// TIA Portal V15.1 export
// export: Created 2024-06-21T08:41:15.2756502Z, ExportSetting WithDefaults, DisplayName Totally Integrated Automation Portal, DisplayVersion V15.1 Update 5, DisplayName TIA Portal Openness, DisplayVersion V15.1 Update 5, DisplayName SINAMICS Startdrive Advanced, DisplayVersion V15.1, DisplayName G130, G150, S120, S150, SINAMICS MV, S210, DisplayVersion V15.1, DisplayName G110M, G120, G120C, G120D, G120P, DisplayVersion V15.1, DisplayName STEP 7 Professional, DisplayVersion V15.1 Update 5, DisplayName STEP 7 Safety, DisplayVersion V15.1, DisplayName WinCC Professional, DisplayVersion V15.1 Update 5, DisplayName SIMATIC Visualization Architect, DisplayVersion V15.1
FUNCTION_BLOCK "LGBChain2W1S-FC302PN"   // FB6603, FBD
TITLE = LGBChain2W1S-FC302PN
{ S7_Optimized_Access := 'FALSE' }
VERSION : 0.1
// stored: AutoNumber false, IsIECCheckEnabled false, SetENOAutomatically False, UDAEnableTagReadback false
   VAR_INPUT
      I_ExitDet { ExternalAccessible := 'False'; ExternalVisible := 'False'; ExternalWritable := 'False'} : Bool;   // Stop Detection set
      I_EntranceDet { ExternalAccessible := 'False'; ExternalVisible := 'False'; ExternalWritable := 'False'} : Bool;   // Stop Detection Reset
      I_StopDetPrev { ExternalAccessible := 'False'; ExternalVisible := 'False'; ExternalWritable := 'False'} : Bool;   // Stop Detection previous conveyor
      I_ChainTensionLDet { ExternalAccessible := 'False'; ExternalVisible := 'False'; ExternalWritable := 'False'} : Bool;   // Chain Tension left detection
      I_ChainTensionRDet { ExternalAccessible := 'False'; ExternalVisible := 'False'; ExternalWritable := 'False'} : Bool;   // Chain Tension Right detection
      I_SlackChainDet { ExternalAccessible := 'False'; ExternalVisible := 'False'; ExternalWritable := 'False'} : Bool;   // Slack Chain detection
      I_TrfInSetBegin { ExternalAccessible := 'False'; ExternalVisible := 'False'; ExternalWritable := 'False'} : Bool;   // Load Begin: condition to start transfer IN set
      I_TrfInSetIntlkOk { ExternalAccessible := 'False'; ExternalVisible := 'False'; ExternalWritable := 'False'} : Bool;   // Transfer IN Interlock Set OK
      I_TrfOutSetBegin { ExternalAccessible := 'False'; ExternalVisible := 'False'; ExternalWritable := 'False'} : Bool;   // Unload Begin: condition to start transfer OUT set
      I_TrfOutSetIntlkOk { ExternalAccessible := 'False'; ExternalVisible := 'False'; ExternalWritable := 'False'} : Bool;   // Transfer Out Interlock Set OK
      I_TrfInSetRdyDlv { ExternalAccessible := 'False'; ExternalVisible := 'False'; ExternalWritable := 'False'} : Bool;   // Ready to deliver: Signal from previous object set
      I_TrfInSetTM { ExternalAccessible := 'False'; ExternalVisible := 'False'; ExternalWritable := 'False'} : Bool;   // Transfer busy signal from previous equipement set
      I_TrfOutSetRdyRcv { ExternalAccessible := 'False'; ExternalVisible := 'False'; ExternalWritable := 'False'} : Bool;   // Ready to Receive: Signal from next object set
      I_TrfOutSetArrived { ExternalAccessible := 'False'; ExternalVisible := 'False'; ExternalWritable := 'False'} : Bool;   // Body Arrived: Signal from next object Set
      I_PBSet { ExternalAccessible := 'False'; ExternalVisible := 'False'; ExternalWritable := 'False'} : Bool;   // Push button for manual movement (on local panel) set
      I_PBReset { ExternalAccessible := 'False'; ExternalVisible := 'False'; ExternalWritable := 'False'} : Bool;   // Push button for manual movement (on local panel) Reset
      I_ManInfeedAllowedSet { ExternalAccessible := 'False'; ExternalVisible := 'False'; ExternalWritable := 'False'} : Bool;   // Manual Infeed Allowed Set (without PushButton)
      I_ManInfeedAllowedRes { ExternalAccessible := 'False'; ExternalVisible := 'False'; ExternalWritable := 'False'} : Bool;   // Manual Infeed Allowed Reset (without PushButton)
      I_MotorProtection { ExternalAccessible := 'False'; ExternalVisible := 'False'; ExternalWritable := 'False'} : Bool;   // Motorprotection
      I_BrakeProtection { ExternalAccessible := 'False'; ExternalVisible := 'False'; ExternalWritable := 'False'} : Bool;   // Brake protection
      I_SafetySwitch { ExternalAccessible := 'False'; ExternalVisible := 'False'; ExternalWritable := 'False'} : Bool;   // Safety switch
      I_ReleaseBrakeMot { ExternalAccessible := 'False'; ExternalVisible := 'False'; ExternalWritable := 'False'} : Bool;   // Release brake motor
      I_SafetyOk { ExternalAccessible := 'False'; ExternalVisible := 'False'; ExternalWritable := 'False'} : Bool;   // Safety Ok
      I_MotionStopOk { ExternalAccessible := 'False'; ExternalVisible := 'False'; ExternalWritable := 'False'} : Bool;   // Safety Ok / The motion stop is Ok
      I_ProductionStop { ExternalAccessible := 'False'; ExternalVisible := 'False'; ExternalWritable := 'False'} : Bool;   // Production Stop
      I_ExtStartConveyor { ExternalAccessible := 'False'; ExternalVisible := 'False'; ExternalWritable := 'False'} : Bool;   // External Start Conveyor
      I_SpeedSetPoint { ExternalAccessible := 'False'; ExternalVisible := 'False'; ExternalWritable := 'False'} : Real;   // Speed set point value motor (cm/min)
      I_ChainEmptyTime { ExternalAccessible := 'False'; ExternalVisible := 'False'; ExternalWritable := 'False'} : DInt;   // Time to empty Chain (Msec)
   END_VAR
   VAR_OUTPUT
      O_Active { ExternalAccessible := 'False'; ExternalVisible := 'False'; ExternalWritable := 'False'} : Bool;   // Chain is Active
      O_TrfInSetRdyRcv { ExternalAccessible := 'False'; ExternalVisible := 'False'; ExternalWritable := 'False'} : Bool;   // Ready to Receive: Signal to previous object set
      O_TrfInSetArrived { ExternalAccessible := 'False'; ExternalVisible := 'False'; ExternalWritable := 'False'} : Bool;   // Body Arrived: Signal to previous object Set
      O_TrfOutSetRdyDlv { ExternalAccessible := 'False'; ExternalVisible := 'False'; ExternalWritable := 'False'} : Bool;   // Ready to Deliver: Signal to next object set
      O_TrfOutSetTM { ExternalAccessible := 'False'; ExternalVisible := 'False'; ExternalWritable := 'False'} : Bool;   // Transfer: Signal to next object set
      O_TrfInSetActive { ExternalAccessible := 'False'; ExternalVisible := 'False'; ExternalWritable := 'False'} : Bool;   // Transfer in set active
      O_TrfInSetFinished { ExternalAccessible := 'False'; ExternalVisible := 'False'; ExternalWritable := 'False'} : Bool;   // Transfer in set finished
      O_TrfOutSetActive { ExternalAccessible := 'False'; ExternalVisible := 'False'; ExternalWritable := 'False'} : Bool;   // Transfer out set active
      O_TrfOutSetFinished { ExternalAccessible := 'False'; ExternalVisible := 'False'; ExternalWritable := 'False'} : Bool;   // Transfer out set finished
      O_LedRoller { ExternalAccessible := 'False'; ExternalVisible := 'False'; ExternalWritable := 'False'} : Bool;   // Led of Chain
      O_SetMotorCmd { ExternalAccessible := 'False'; ExternalVisible := 'False'; ExternalWritable := 'False'} : Bool;   // High Speed Set Command from function after Interlock
      O_ResMotorCmd { ExternalAccessible := 'False'; ExternalVisible := 'False'; ExternalWritable := 'False'} : Bool;   // High speed Reset Command from function after Interlock
      O_AlarmABCondition { ExternalAccessible := 'False'; ExternalVisible := 'False'; ExternalWritable := 'False'} : Bool;   // Alarm AB Condition
      O_AlarmA { ExternalAccessible := 'False'; ExternalVisible := 'False'; ExternalWritable := 'False'} : Bool;   // Alarm A
      O_AlarmB { ExternalAccessible := 'False'; ExternalVisible := 'False'; ExternalWritable := 'False'} : Bool;   // Alarm B
      O_AlarmC { ExternalAccessible := 'False'; ExternalVisible := 'False'; ExternalWritable := 'False'} : Bool;   // Alarm C
      O_AlarmD { ExternalAccessible := 'False'; ExternalVisible := 'False'; ExternalWritable := 'False'} : Bool;   // Alarm D
      O_Occupied { ExternalAccessible := 'False'; ExternalVisible := 'False'; ExternalWritable := 'False'} : Bool;   // Chain Occupied
      O_ActualSpeed { ExternalAccessible := 'False'; ExternalVisible := 'False'; ExternalWritable := 'False'} : Int;   // Actual speed value motor (cm/min)
      O_ActualCurrent { ExternalAccessible := 'False'; ExternalVisible := 'False'; ExternalWritable := 'False'} : Real;   // Actual Current value motor (A)
      H_AlarmDWord { ExternalAccessible := 'False'; ExternalVisible := 'False'; ExternalWritable := 'False'} : DWord;   // HMI Animation
   END_VAR
   VAR_IN_OUT
      C_TimeCheckSpeedOK { ExternalAccessible := 'False'; ExternalVisible := 'False'; ExternalWritable := 'False'} : DInt := 2000;   // Time check speed OK
      IO_Modes : "Modes";   // Modes
      H_HMI : "H_HMI";   // Animation
      "H_GBChain2W1S-FC302PN" : "H_GBChain2W1S-FC302PN";   // Animation
      C_Config : "RollerConvConfig";   // Config
   END_VAR
   VAR DB_SPECIFIC
      H_FncSelInHMI { ExternalAccessible := 'False'; ExternalVisible := 'False'; ExternalWritable := 'False'} : Bool;
      AB_ChainTensionLAlm { ExternalAccessible := 'False'; ExternalVisible := 'False'; ExternalWritable := 'False'} : Bool;   // Alarm Chain Tension Left
      AB_ChainTensionRAlm { ExternalAccessible := 'False'; ExternalVisible := 'False'; ExternalWritable := 'False'} : Bool;   // Alarm Chain Tension Right
      AB_SlackChainAlm { ExternalAccessible := 'False'; ExternalVisible := 'False'; ExternalWritable := 'False'} : Bool;   // Alarm Slack Chain
      AC_TrfOutSetOverTime { ExternalAccessible := 'False'; ExternalVisible := 'False'; ExternalWritable := 'False'} : Bool;   // Timeout Transport Out Set
      AD_TrfOutSetInterlock { ExternalAccessible := 'False'; ExternalVisible := 'False'; ExternalWritable := 'False'} : Bool;   // Interlock Not Ok Transport Out Set
      AD_TrfInSetInterlock { ExternalAccessible := 'False'; ExternalVisible := 'False'; ExternalWritable := 'False'} : Bool;   // Interlock Not Ok Transport In Set
      AA_BusFault { ExternalAccessible := 'False'; ExternalVisible := 'False'; ExternalWritable := 'False'} : Bool;   // Drive Bus Fault
      AA_MotorProtector { ExternalAccessible := 'False'; ExternalVisible := 'False'; ExternalWritable := 'False'} : Bool;   // Motor Protection Tripped
      AA_BrakeProtection { ExternalAccessible := 'False'; ExternalVisible := 'False'; ExternalWritable := 'False'} : Bool;   // Brake Protection Tripped
      AA_SafetySwitch { ExternalAccessible := 'False'; ExternalVisible := 'False'; ExternalWritable := 'False'} : Bool;   // Safety Switch Not Ok
      AD_WarningFrqcnvMot { ExternalAccessible := 'False'; ExternalVisible := 'False'; ExternalWritable := 'False'} : Bool;   // Frequency Control FC302 Warning motor
      AB_AlarmFrqcnvMot { ExternalAccessible := 'False'; ExternalVisible := 'False'; ExternalWritable := 'False'} : Bool;   // Frequency Control FC302 Alarm motor
      AB_CurrentSensorAlm { ExternalAccessible := 'False'; ExternalVisible := 'False'; ExternalWritable := 'False'} : Bool;   // Over Current Motor
      AB_OverCurrentHHAlm { ExternalAccessible := 'False'; ExternalVisible := 'False'; ExternalWritable := 'False'} : Bool;   // Over Current Motor
      AB_OverCurrentHAlm { ExternalAccessible := 'False'; ExternalVisible := 'False'; ExternalWritable := 'False'} : Bool;   // Over Current Motor
      AB_OverCurrentLAlm { ExternalAccessible := 'False'; ExternalVisible := 'False'; ExternalWritable := 'False'} : Bool;   // Over Current Motor
      AB_OverCurrentLLAlm { ExternalAccessible := 'False'; ExternalVisible := 'False'; ExternalWritable := 'False'} : Bool;   // Over Current Motor
      AD_MotionStop { ExternalAccessible := 'False'; ExternalVisible := 'False'; ExternalWritable := 'False'} : Bool;   // Motion Stop
      AC_ConfigCalibrationAlm { ExternalAccessible := 'False'; ExternalVisible := 'False'; ExternalWritable := 'False'} : Bool;   // The Config values for Alarm Transfer time must be ALL zero or ALL different from zero
      AD_CalibrationSetWarn { ExternalAccessible := 'False'; ExternalVisible := 'False'; ExternalWritable := 'False'} : Bool;   // No High speed selected so Calibration is not possible for SET direction
      SafetyOk { ExternalAccessible := 'False'; ExternalVisible := 'False'; ExternalWritable := 'False'} : Bool;   // Safety Ok
      OverCurrentHAlmCond { ExternalAccessible := 'False'; ExternalVisible := 'False'; ExternalWritable := 'False'} : Bool;   // Over Current Motor
      ChainTensionLAlmCond { ExternalAccessible := 'False'; ExternalVisible := 'False'; ExternalWritable := 'False'} : Bool;   // Alarm Chain Tension Left
      ChainTensionRAlmCond { ExternalAccessible := 'False'; ExternalVisible := 'False'; ExternalWritable := 'False'} : Bool;   // Alarm Chain Tension Right
      SlackChainAlmCond { ExternalAccessible := 'False'; ExternalVisible := 'False'; ExternalWritable := 'False'} : Bool;   // Alarm Slack Chain
      MotorLoopActive { ExternalAccessible := 'False'; ExternalVisible := 'False'; ExternalWritable := 'False'} : Bool;   // Motor Loop Active
      TrfInfeedHoldSet { ExternalAccessible := 'False'; ExternalVisible := 'False'; ExternalWritable := 'False'} : Bool;   // Transfer infeed hold set direction
      TrfOutSetCmd { ExternalAccessible := 'False'; ExternalVisible := 'False'; ExternalWritable := 'False'} : Bool;   // Command after Interlock to Motor set
      TrfOutfeedHoldSet { ExternalAccessible := 'False'; ExternalVisible := 'False'; ExternalWritable := 'False'} : Bool;   // Transfer outfeed hold set direction
      TrfInSetCmd { ExternalAccessible := 'False'; ExternalVisible := 'False'; ExternalWritable := 'False'} : Bool;   // Command after Interlock to Motor set
      MotorCmdSet { ExternalAccessible := 'False'; ExternalVisible := 'False'; ExternalWritable := 'False'} : Bool;   // Command to Motorloop High Speed Set
      MotorCmdRes { ExternalAccessible := 'False'; ExternalVisible := 'False'; ExternalWritable := 'False'} : Bool;   // Command to Motorloop High Speed Reset
      TrfInSetActive { ExternalAccessible := 'False'; ExternalVisible := 'False'; ExternalWritable := 'False'} : Bool;   // Load: Active (set)
      TrfOutSetActive { ExternalAccessible := 'False'; ExternalVisible := 'False'; ExternalWritable := 'False'} : Bool;   // Unload: active (set)
      TrfOutSetFinished { ExternalAccessible := 'False'; ExternalVisible := 'False'; ExternalWritable := 'False'} : Bool;   // Unload: finished (set)
      AlarmA { ExternalAccessible := 'False'; ExternalVisible := 'False'; ExternalWritable := 'False'} : Bool;   // Alarm A
      AlarmB { ExternalAccessible := 'False'; ExternalVisible := 'False'; ExternalWritable := 'False'} : Bool;   // Alarm B
      AlarmC { ExternalAccessible := 'False'; ExternalVisible := 'False'; ExternalWritable := 'False'} : Bool;   // Alarm C
      AlarmD { ExternalAccessible := 'False'; ExternalVisible := 'False'; ExternalWritable := 'False'} : Bool;   // Alarm D
      ManLowSpdSel { ExternalAccessible := 'False'; ExternalVisible := 'False'; ExternalWritable := 'False'} : Bool;   // Low speed Selected in manual
      TrfOutSetRdyDlv { ExternalAccessible := 'False'; ExternalVisible := 'False'; ExternalWritable := 'False'} : Bool;   // Ready to Deliver: Signal to next object set
      TrfOutSetTM { ExternalAccessible := 'False'; ExternalVisible := 'False'; ExternalWritable := 'False'} : Bool;   // Transfer : Signal transfer memory to next object set
      TrfInSetTrfOutSetTM { ExternalAccessible := 'False'; ExternalVisible := 'False'; ExternalWritable := 'False'} : Bool;   // Transfer memory set
      TrfInSetRdyRcv { ExternalAccessible := 'False'; ExternalVisible := 'False'; ExternalWritable := 'False'} : Bool;   // Ready to Receive: Signal to previous object set
      TrfInSetArrived { ExternalAccessible := 'False'; ExternalVisible := 'False'; ExternalWritable := 'False'} : Bool;   // Body Arrived: Signal to previous object Set
      TrfInSetFinished { ExternalAccessible := 'False'; ExternalVisible := 'False'; ExternalWritable := 'False'} : Bool;   // Body Arrived: Signal to TrfOut module set (Reset TrfOutCmd)
      StopTrfOutSetCmd { ExternalAccessible := 'False'; ExternalVisible := 'False'; ExternalWritable := 'False'} : Bool;   // Body Arrived: Signal to previous object Set
      MotorLoopAlmCond { ExternalAccessible := 'False'; ExternalVisible := 'False'; ExternalWritable := 'False'} : Bool;   // Motor loop Alarm condition
      TrfOutSetAlmCond { ExternalAccessible := 'False'; ExternalVisible := 'False'; ExternalWritable := 'False'} : Bool;   // TrfOut set Alarm condition
      FrqReadyForOperationMot { ExternalAccessible := 'False'; ExternalVisible := 'False'; ExternalWritable := 'False'} : Bool;   // Fb motor is ready to operate motor
      ReleaseBrakeMot { ExternalAccessible := 'False'; ExternalVisible := 'False'; ExternalWritable := 'False'} : Bool;   // Req to release brake motor
      ChainStop { ExternalAccessible := 'False'; ExternalVisible := 'False'; ExternalWritable := 'False'} : Bool;   // Chain stop Productions Stop
      DlvSaturation { ExternalAccessible := 'False'; ExternalVisible := 'False'; ExternalWritable := 'False'} : Bool;   // Saturation for the diliver tranfer
      AlarmABCondition { ExternalAccessible := 'False'; ExternalVisible := 'False'; ExternalWritable := 'False'} : Bool;   // Alarm AB Condition
      HighSpeedMot { ExternalAccessible := 'False'; ExternalVisible := 'False'; ExternalWritable := 'False'} : Real;   // High speed Value (set-up %) Motor
      ActualSpeed { ExternalAccessible := 'False'; ExternalVisible := 'False'; ExternalWritable := 'False'} : Real;   // Actual Speed in % from FC302
      ChainEmpty { ExternalAccessible := 'False'; ExternalVisible := 'False'; ExternalWritable := 'False'} : Bool;   // Chain is Empty
      OverCurrAlarm { ExternalAccessible := 'False'; ExternalVisible := 'False'; ExternalWritable := 'False'} : Bool;
      AnInput { ExternalAccessible := 'False'; ExternalVisible := 'False'; ExternalWritable := 'False'} : Real;   // Actual Current
   END_VAR
   VAR
      _ChainEmptyTimer { ExternalAccessible := 'False'; ExternalVisible := 'False'; ExternalWritable := 'False'} : "LTimer";   // Timer
      _LTrfInSet { ExternalAccessible := 'False'; ExternalVisible := 'False'; ExternalWritable := 'False'} : "LGBTrfIn";   // FB
      _LTrfOutSet { ExternalAccessible := 'False'; ExternalVisible := 'False'; ExternalWritable := 'False'} : "LGBTrfOut";   // FB
      _Motor { ExternalAccessible := 'False'; ExternalVisible := 'False'; ExternalWritable := 'False'} : "LGBMotor2W2S-FC302PN";
      _MotorCurrent : "LAnInput6Lim";
      _ChainTensionLeft { ExternalAccessible := 'False'; ExternalVisible := 'False'; ExternalWritable := 'False'} : "L1AlarmMultiIn";
      _ChainTensionRight { ExternalAccessible := 'False'; ExternalVisible := 'False'; ExternalWritable := 'False'} : "L1AlarmMultiIn";
      _ChainSlack { ExternalAccessible := 'False'; ExternalVisible := 'False'; ExternalWritable := 'False'} : "L1AlarmMultiIn";
   END_VAR
   VAR DB_SPECIFIC
      Reset_TP { ExternalAccessible := 'False'; ExternalVisible := 'False'; ExternalWritable := 'False'} : TP_TIME;
   END_VAR
   VAR_TEMP
      H_HMITrfInSet : "H_HMI";   // Temp
      H_HMITrfOutSet : "H_HMI";   // Temp
      H_HMIMotor : "H_HMI";   // Temp
   END_VAR
   VAR_TEMP   // added for the SCL form of the ladder/FBD networks
      _w1 : Bool;
   END_VAR
BEGIN

REGION Network 1: **** 1 - Inputs **** Safety Ok
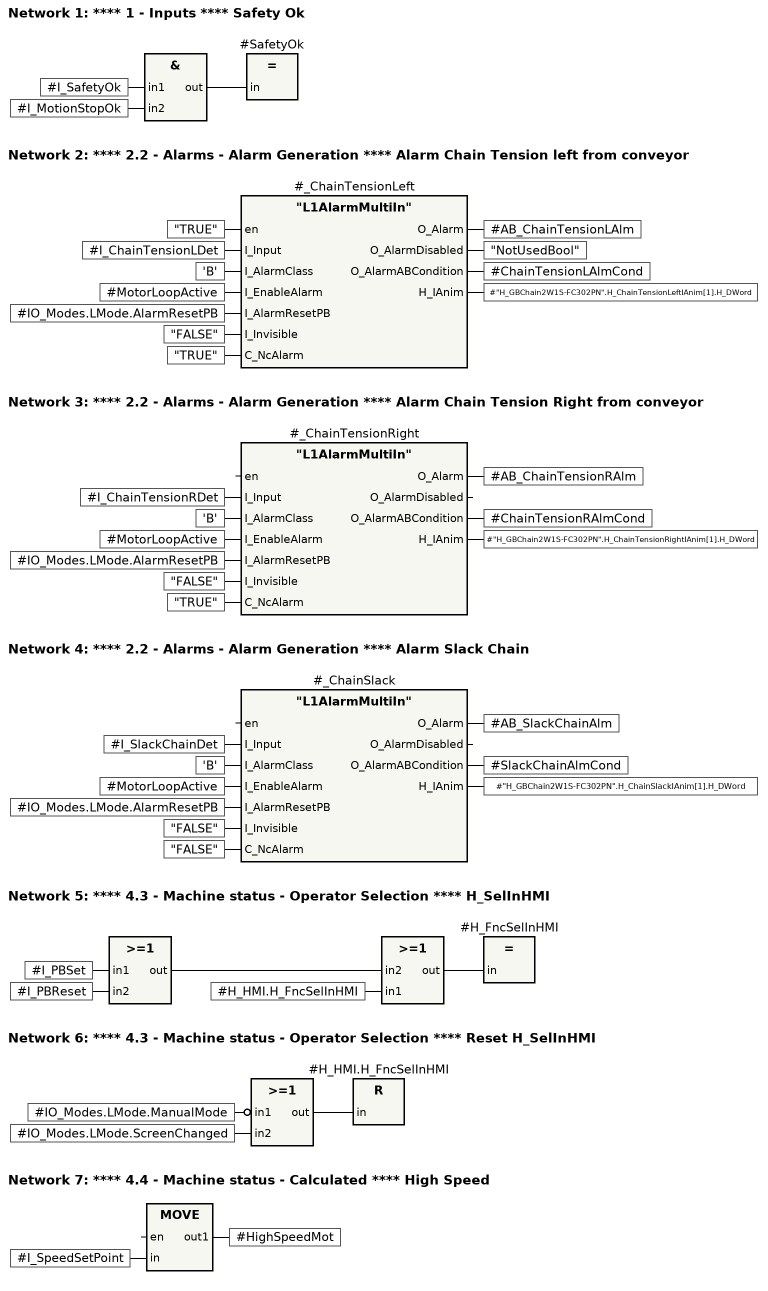
   #SafetyOk := #I_SafetyOk AND #I_MotionStopOk;
END_REGION

REGION Network 2: **** 2.2 - Alarms - Alarm Generation **** Alarm Chain Tension left from conveyor
   // Alarm Chain tension conveyor
   IF "TRUE" THEN
       #_ChainTensionLeft(I_Input := #I_ChainTensionLDet,   // "L1AlarmMultiIn"
                          I_AlarmClass := 'B',
                          I_EnableAlarm := #MotorLoopActive,
                          I_AlarmResetPB := #IO_Modes.LMode.AlarmResetPB,
                          I_Invisible := "FALSE",
                          C_NcAlarm := "TRUE",
                          O_Alarm => #AB_ChainTensionLAlm,
                          O_AlarmDisabled => "NotUsedBool",
                          O_AlarmABCondition => #ChainTensionLAlmCond,
                          H_IAnim => #"H_GBChain2W1S-FC302PN".H_ChainTensionLeftIAnim[1].H_DWord);
   END_IF;
END_REGION

REGION Network 3: **** 2.2 - Alarms - Alarm Generation **** Alarm Chain Tension Right from conveyor
   // Alarm Chain tension conveyor
   #_ChainTensionRight(I_Input := #I_ChainTensionRDet,   // "L1AlarmMultiIn"
                       I_AlarmClass := 'B',
                       I_EnableAlarm := #MotorLoopActive,
                       I_AlarmResetPB := #IO_Modes.LMode.AlarmResetPB,
                       I_Invisible := "FALSE",
                       C_NcAlarm := "TRUE",
                       O_Alarm => #AB_ChainTensionRAlm,
                       O_AlarmABCondition => #ChainTensionRAlmCond,
                       H_IAnim => #"H_GBChain2W1S-FC302PN".H_ChainTensionRightIAnim[1].H_DWord);
END_REGION

REGION Network 4: **** 2.2 - Alarms - Alarm Generation **** Alarm Slack Chain
   // Alarm Slack Chain
   #_ChainSlack(I_Input := #I_SlackChainDet,   // "L1AlarmMultiIn"
                I_AlarmClass := 'B',
                I_EnableAlarm := #MotorLoopActive,
                I_AlarmResetPB := #IO_Modes.LMode.AlarmResetPB,
                I_Invisible := "FALSE",
                C_NcAlarm := "FALSE",
                O_Alarm => #AB_SlackChainAlm,
                O_AlarmABCondition => #SlackChainAlmCond,
                H_IAnim => #"H_GBChain2W1S-FC302PN".H_ChainSlackIAnim[1].H_DWord);
END_REGION

REGION Network 5: **** 4.3 - Machine status - Operator Selection **** H_SelInHMI
   #H_FncSelInHMI := #I_PBSet OR #I_PBReset OR #H_HMI.H_FncSelInHMI;
END_REGION

REGION Network 6: **** 4.3 - Machine status - Operator Selection **** Reset H_SelInHMI
   // Reset H_SelInHMI
   IF NOT #IO_Modes.LMode.ManualMode OR #IO_Modes.LMode.ScreenChanged THEN
       #H_HMI.H_FncSelInHMI := FALSE;
   END_IF;
END_REGION

REGION Network 7: **** 4.4 - Machine status - Calculated **** High Speed
   #HighSpeedMot := #I_SpeedSetPoint;
END_REGION

REGION Network 8: **** 4.4 - Machine status - Calculated **** High Speed Motor to high
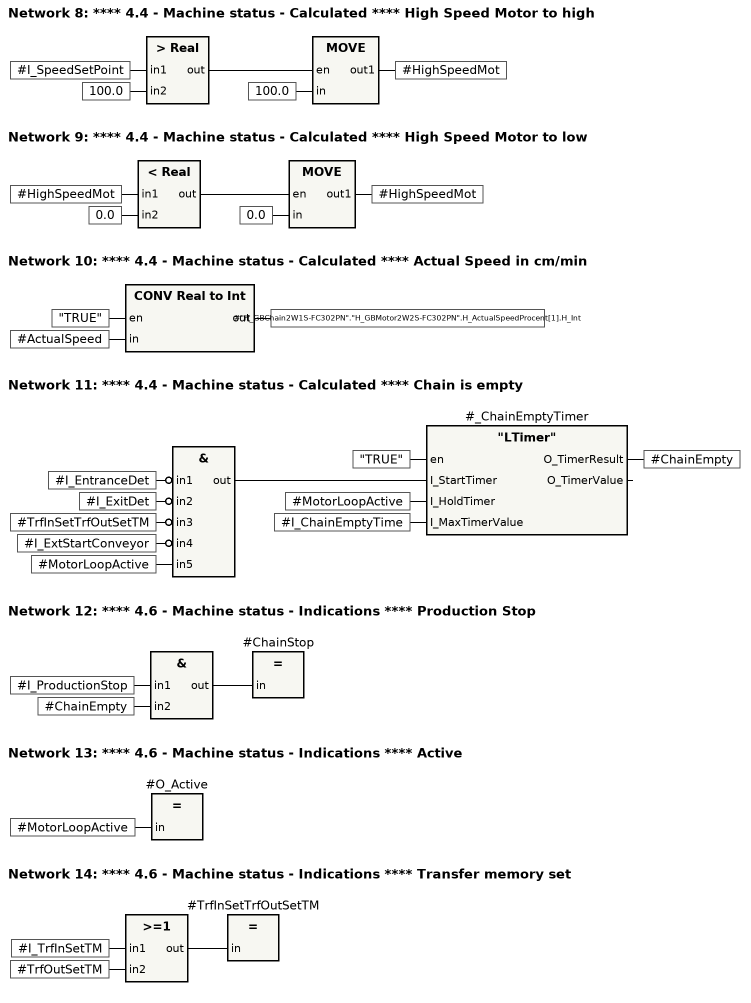
   IF #I_SpeedSetPoint > 100.0 THEN #HighSpeedMot := 100.0; END_IF;
END_REGION

REGION Network 9: **** 4.4 - Machine status - Calculated **** High Speed Motor to low
   IF #HighSpeedMot < 0.0 THEN #HighSpeedMot := 0.0; END_IF;
END_REGION

REGION Network 10: **** 4.4 - Machine status - Calculated **** Actual Speed in cm/min
   // Actual Speed in cm/min
   IF "TRUE" THEN
       #"H_GBChain2W1S-FC302PN"."H_GBMotor2W2S-FC302PN".H_ActualSpeedProcent[1].H_Int := REAL_TO_INT(#ActualSpeed);
   END_IF;
END_REGION

REGION Network 11: **** 4.4 - Machine status - Calculated **** Chain is empty
   // Chain is empty when chain is running and no detection is activated during the preset time
   IF "TRUE" THEN
       #_ChainEmptyTimer(I_StartTimer := NOT #I_EntranceDet AND NOT #I_ExitDet AND NOT #TrfInSetTrfOutSetTM AND NOT #I_ExtStartConveyor AND #MotorLoopActive,   // "LTimer"
                         I_HoldTimer := #MotorLoopActive,
                         I_MaxTimerValue := #I_ChainEmptyTime,
                         O_TimerResult => #ChainEmpty);
   END_IF;
END_REGION

REGION Network 12: **** 4.6 - Machine status - Indications **** Production Stop
   #ChainStop := #I_ProductionStop AND #ChainEmpty;
END_REGION

REGION Network 13: **** 4.6 - Machine status - Indications **** Active
   // Active
   #O_Active := #MotorLoopActive;
END_REGION

REGION Network 14: **** 4.6 - Machine status - Indications **** Transfer memory set
   // Transfer memory set
   #TrfInSetTrfOutSetTM := #I_TrfInSetTM OR #TrfOutSetTM;
END_REGION

REGION Network 15: **** 4.6 - Machine Status - Indication **** Entrance Det
   // Entrance Det
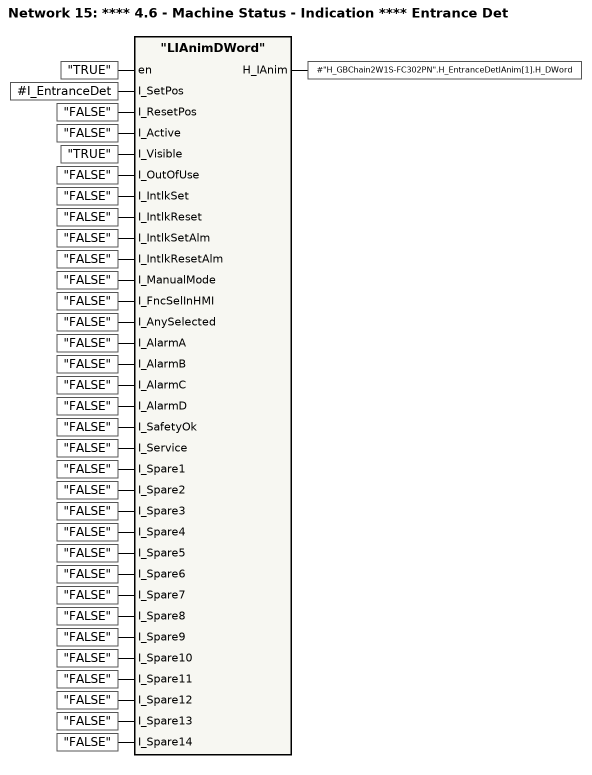
   IF "TRUE" THEN
       "LIAnimDWord"(I_SetPos := #I_EntranceDet,
                     I_ResetPos := "FALSE",
                     I_Active := "FALSE",
                     I_Visible := "TRUE",
                     I_OutOfUse := "FALSE",
                     I_IntlkSet := "FALSE",
                     I_IntlkReset := "FALSE",
                     I_IntlkSetAlm := "FALSE",
                     I_IntlkResetAlm := "FALSE",
                     I_ManualMode := "FALSE",
                     I_FncSelInHMI := "FALSE",
                     I_AnySelected := "FALSE",
                     I_AlarmA := "FALSE",
                     I_AlarmB := "FALSE",
                     I_AlarmC := "FALSE",
                     I_AlarmD := "FALSE",
                     I_SafetyOk := "FALSE",
                     I_Service := "FALSE",
                     I_Spare1 := "FALSE",
                     I_Spare2 := "FALSE",
                     I_Spare3 := "FALSE",
                     I_Spare4 := "FALSE",
                     I_Spare5 := "FALSE",
                     I_Spare6 := "FALSE",
                     I_Spare7 := "FALSE",
                     I_Spare8 := "FALSE",
                     I_Spare9 := "FALSE",
                     I_Spare10 := "FALSE",
                     I_Spare11 := "FALSE",
                     I_Spare12 := "FALSE",
                     I_Spare13 := "FALSE",
                     I_Spare14 := "FALSE",
                     H_IAnim => #"H_GBChain2W1S-FC302PN".H_EntranceDetIAnim[1].H_DWord);
   END_IF;
END_REGION

REGION Network 16: **** 4.6 - Machine Status - Indication **** Exit Det
   // Exit Det
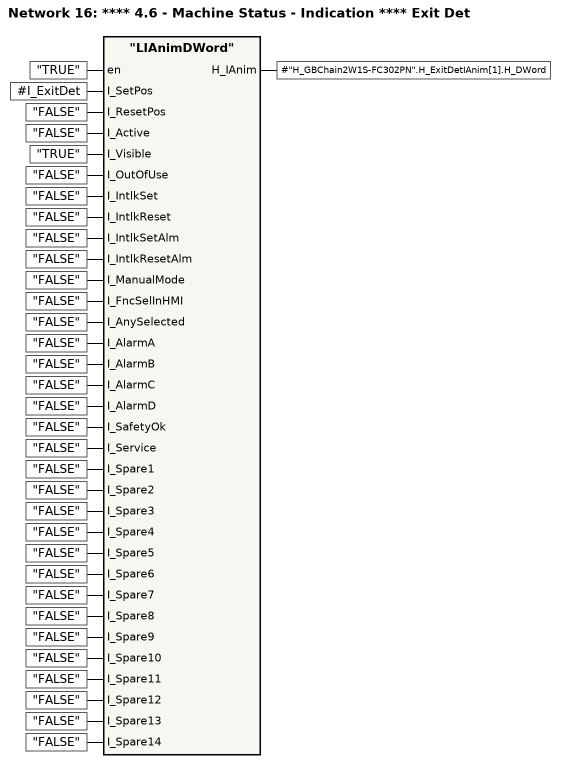
   IF "TRUE" THEN
       "LIAnimDWord"(I_SetPos := #I_ExitDet,
                     I_ResetPos := "FALSE",
                     I_Active := "FALSE",
                     I_Visible := "TRUE",
                     I_OutOfUse := "FALSE",
                     I_IntlkSet := "FALSE",
                     I_IntlkReset := "FALSE",
                     I_IntlkSetAlm := "FALSE",
                     I_IntlkResetAlm := "FALSE",
                     I_ManualMode := "FALSE",
                     I_FncSelInHMI := "FALSE",
                     I_AnySelected := "FALSE",
                     I_AlarmA := "FALSE",
                     I_AlarmB := "FALSE",
                     I_AlarmC := "FALSE",
                     I_AlarmD := "FALSE",
                     I_SafetyOk := "FALSE",
                     I_Service := "FALSE",
                     I_Spare1 := "FALSE",
                     I_Spare2 := "FALSE",
                     I_Spare3 := "FALSE",
                     I_Spare4 := "FALSE",
                     I_Spare5 := "FALSE",
                     I_Spare6 := "FALSE",
                     I_Spare7 := "FALSE",
                     I_Spare8 := "FALSE",
                     I_Spare9 := "FALSE",
                     I_Spare10 := "FALSE",
                     I_Spare11 := "FALSE",
                     I_Spare12 := "FALSE",
                     I_Spare13 := "FALSE",
                     I_Spare14 := "FALSE",
                     H_IAnim => #"H_GBChain2W1S-FC302PN".H_ExitDetIAnim[1].H_DWord);
   END_IF;
END_REGION

REGION Network 17: **** 4.6 - Machine Status - Indication **** Icon Animation
   // Icon Animation
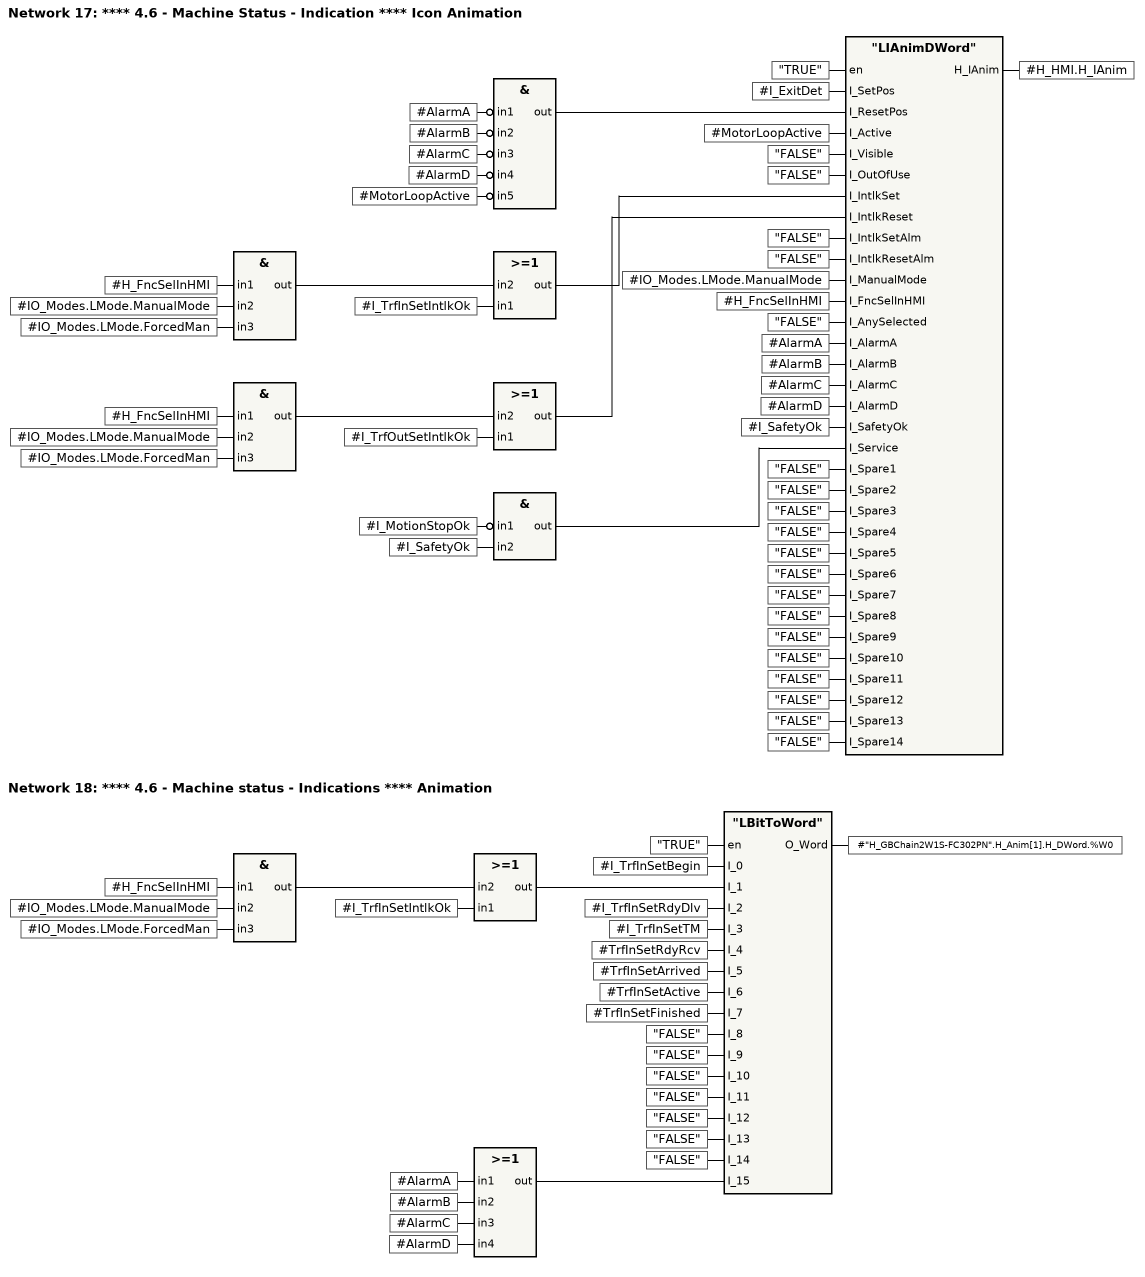
   IF "TRUE" THEN
       "LIAnimDWord"(I_SetPos := #I_ExitDet,
                     I_ResetPos := NOT #AlarmA AND NOT #AlarmB AND NOT #AlarmC AND NOT #AlarmD AND NOT #MotorLoopActive,
                     I_Active := #MotorLoopActive,
                     I_Visible := "FALSE",
                     I_OutOfUse := "FALSE",
                     I_IntlkSet := (#H_FncSelInHMI AND #IO_Modes.LMode.ManualMode AND #IO_Modes.LMode.ForcedMan) OR #I_TrfInSetIntlkOk,
                     I_IntlkReset := (#H_FncSelInHMI AND #IO_Modes.LMode.ManualMode AND #IO_Modes.LMode.ForcedMan) OR #I_TrfOutSetIntlkOk,
                     I_IntlkSetAlm := "FALSE",
                     I_IntlkResetAlm := "FALSE",
                     I_ManualMode := #IO_Modes.LMode.ManualMode,
                     I_FncSelInHMI := #H_FncSelInHMI,
                     I_AnySelected := "FALSE",
                     I_AlarmA := #AlarmA,
                     I_AlarmB := #AlarmB,
                     I_AlarmC := #AlarmC,
                     I_AlarmD := #AlarmD,
                     I_SafetyOk := #I_SafetyOk,
                     I_Service := NOT #I_MotionStopOk AND #I_SafetyOk,
                     I_Spare1 := "FALSE",
                     I_Spare2 := "FALSE",
                     I_Spare3 := "FALSE",
                     I_Spare4 := "FALSE",
                     I_Spare5 := "FALSE",
                     I_Spare6 := "FALSE",
                     I_Spare7 := "FALSE",
                     I_Spare8 := "FALSE",
                     I_Spare9 := "FALSE",
                     I_Spare10 := "FALSE",
                     I_Spare11 := "FALSE",
                     I_Spare12 := "FALSE",
                     I_Spare13 := "FALSE",
                     I_Spare14 := "FALSE",
                     H_IAnim => #H_HMI.H_IAnim);
   END_IF;
END_REGION

REGION Network 18: **** 4.6 - Machine status - Indications **** Animation
   // Animation
   IF "TRUE" THEN
       "LBitToWord"(I_0 := #I_TrfInSetBegin,
                    I_1 := (#H_FncSelInHMI AND #IO_Modes.LMode.ManualMode AND #IO_Modes.LMode.ForcedMan) OR #I_TrfInSetIntlkOk,
                    I_2 := #I_TrfInSetRdyDlv,
                    I_3 := #I_TrfInSetTM,
                    I_4 := #TrfInSetRdyRcv,
                    I_5 := #TrfInSetArrived,
                    I_6 := #TrfInSetActive,
                    I_7 := #TrfInSetFinished,
                    I_8 := "FALSE",
                    I_9 := "FALSE",
                    I_10 := "FALSE",
                    I_11 := "FALSE",
                    I_12 := "FALSE",
                    I_13 := "FALSE",
                    I_14 := "FALSE",
                    I_15 := #AlarmA OR #AlarmB OR #AlarmC OR #AlarmD,
                    O_Word => #"H_GBChain2W1S-FC302PN".H_Anim[1].H_DWord.%W0);
   END_IF;
END_REGION

REGION Network 19: **** 4.6 - Machine status - Indications **** Animation
   // Animation
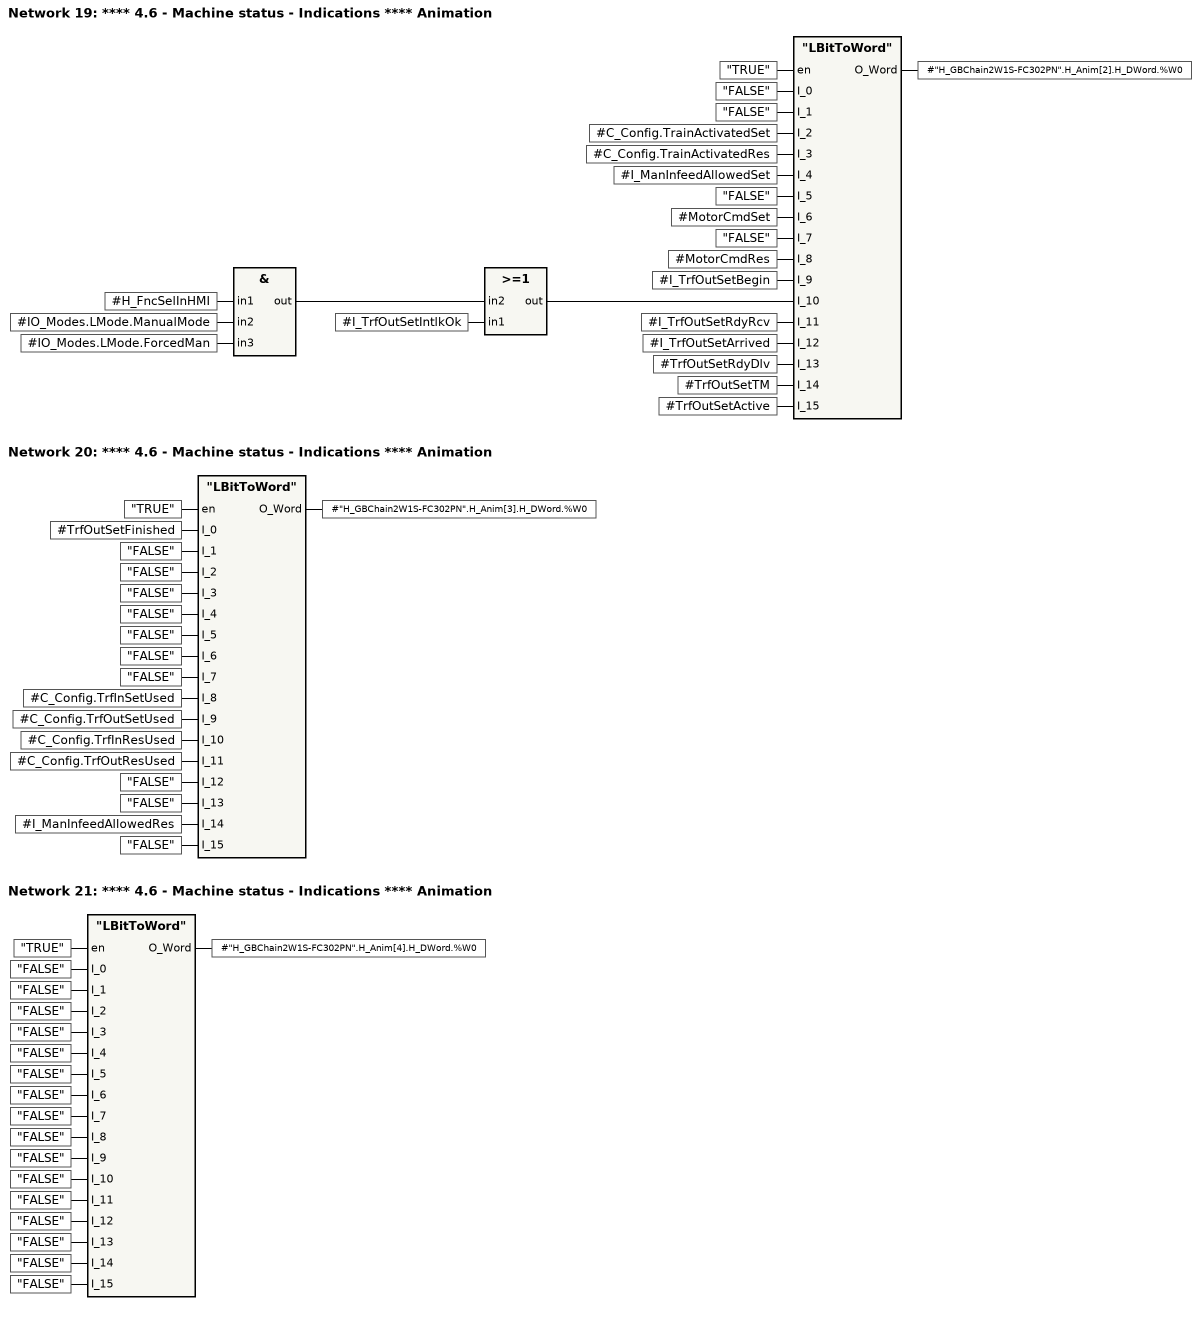
   IF "TRUE" THEN
       "LBitToWord"(I_0 := "FALSE",
                    I_1 := "FALSE",
                    I_2 := #C_Config.TrainActivatedSet,
                    I_3 := #C_Config.TrainActivatedRes,
                    I_4 := #I_ManInfeedAllowedSet,
                    I_5 := "FALSE",
                    I_6 := #MotorCmdSet,
                    I_7 := "FALSE",
                    I_8 := #MotorCmdRes,
                    I_9 := #I_TrfOutSetBegin,
                    I_10 := (#H_FncSelInHMI AND #IO_Modes.LMode.ManualMode AND #IO_Modes.LMode.ForcedMan) OR #I_TrfOutSetIntlkOk,
                    I_11 := #I_TrfOutSetRdyRcv,
                    I_12 := #I_TrfOutSetArrived,
                    I_13 := #TrfOutSetRdyDlv,
                    I_14 := #TrfOutSetTM,
                    I_15 := #TrfOutSetActive,
                    O_Word => #"H_GBChain2W1S-FC302PN".H_Anim[2].H_DWord.%W0);
   END_IF;
END_REGION

REGION Network 20: **** 4.6 - Machine status - Indications **** Animation
   // Animation
   IF "TRUE" THEN
       "LBitToWord"(I_0 := #TrfOutSetFinished,
                    I_1 := "FALSE",
                    I_2 := "FALSE",
                    I_3 := "FALSE",
                    I_4 := "FALSE",
                    I_5 := "FALSE",
                    I_6 := "FALSE",
                    I_7 := "FALSE",
                    I_8 := #C_Config.TrfInSetUsed,
                    I_9 := #C_Config.TrfOutSetUsed,
                    I_10 := #C_Config.TrfInResUsed,
                    I_11 := #C_Config.TrfOutResUsed,
                    I_12 := "FALSE",
                    I_13 := "FALSE",
                    I_14 := #I_ManInfeedAllowedRes,
                    I_15 := "FALSE",
                    O_Word => #"H_GBChain2W1S-FC302PN".H_Anim[3].H_DWord.%W0);
   END_IF;
END_REGION

REGION Network 21: **** 4.6 - Machine status - Indications **** Animation
   // Animation
   IF "TRUE" THEN
       "LBitToWord"(I_0 := "FALSE",
                    I_1 := "FALSE",
                    I_2 := "FALSE",
                    I_3 := "FALSE",
                    I_4 := "FALSE",
                    I_5 := "FALSE",
                    I_6 := "FALSE",
                    I_7 := "FALSE",
                    I_8 := "FALSE",
                    I_9 := "FALSE",
                    I_10 := "FALSE",
                    I_11 := "FALSE",
                    I_12 := "FALSE",
                    I_13 := "FALSE",
                    I_14 := "FALSE",
                    I_15 := "FALSE",
                    O_Word => #"H_GBChain2W1S-FC302PN".H_Anim[4].H_DWord.%W0);
   END_IF;
END_REGION

REGION Network 22: **** 7.1 - Submodule - Non-Machine **** Analoge Input Motor Current
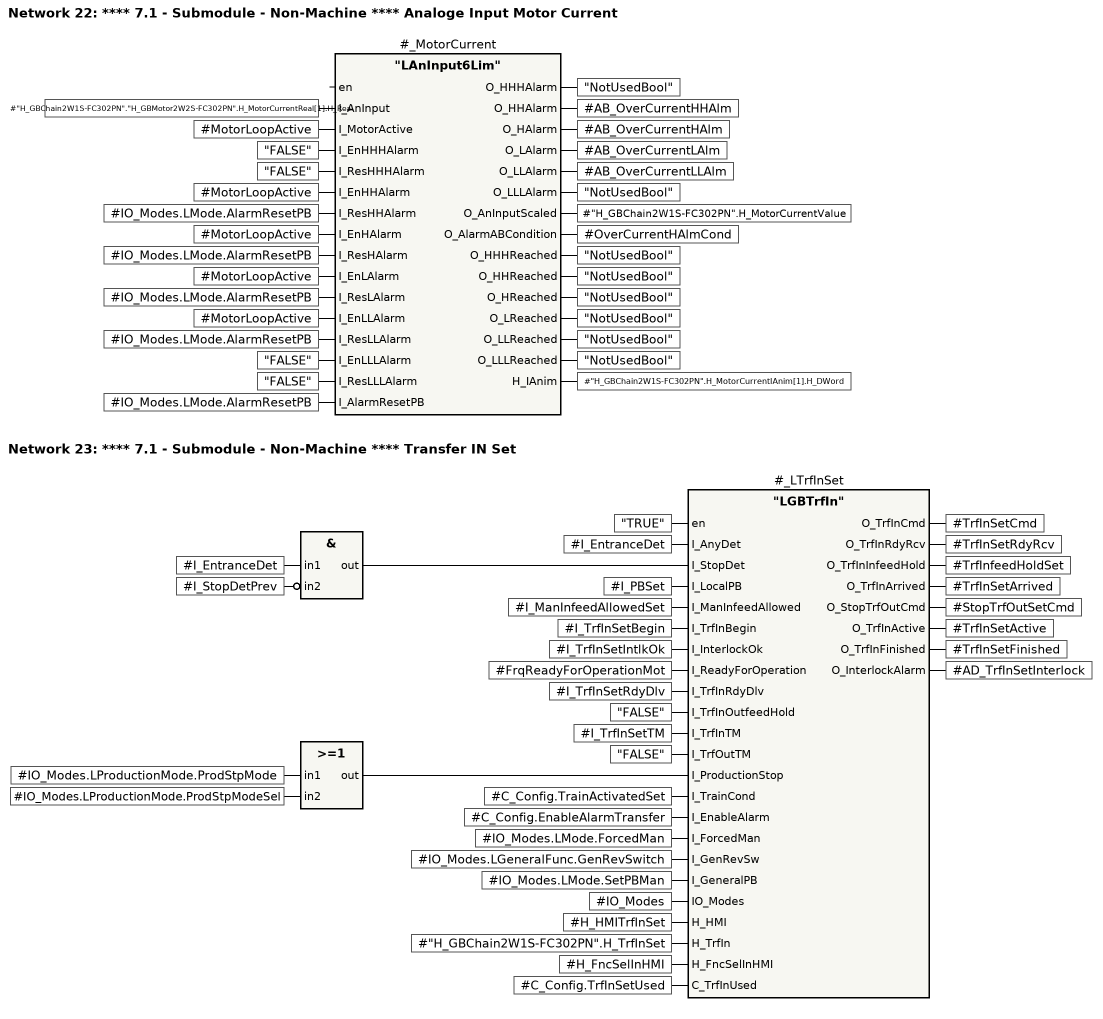
   #_MotorCurrent(I_AnInput := #"H_GBChain2W1S-FC302PN"."H_GBMotor2W2S-FC302PN".H_MotorCurrentReal[1].H_Real,   // "LAnInput6Lim"
                  I_MotorActive := #MotorLoopActive,
                  I_EnHHHAlarm := "FALSE",
                  I_ResHHHAlarm := "FALSE",
                  I_EnHHAlarm := #MotorLoopActive,
                  I_ResHHAlarm := #IO_Modes.LMode.AlarmResetPB,
                  I_EnHAlarm := #MotorLoopActive,
                  I_ResHAlarm := #IO_Modes.LMode.AlarmResetPB,
                  I_EnLAlarm := #MotorLoopActive,
                  I_ResLAlarm := #IO_Modes.LMode.AlarmResetPB,
                  I_EnLLAlarm := #MotorLoopActive,
                  I_ResLLAlarm := #IO_Modes.LMode.AlarmResetPB,
                  I_EnLLLAlarm := "FALSE",
                  I_ResLLLAlarm := "FALSE",
                  I_AlarmResetPB := #IO_Modes.LMode.AlarmResetPB,
                  O_HHHAlarm => "NotUsedBool",
                  O_HHAlarm => #AB_OverCurrentHHAlm,
                  O_HAlarm => #AB_OverCurrentHAlm,
                  O_LAlarm => #AB_OverCurrentLAlm,
                  O_LLAlarm => #AB_OverCurrentLLAlm,
                  O_LLLAlarm => "NotUsedBool",
                  O_AnInputScaled => #"H_GBChain2W1S-FC302PN".H_MotorCurrentValue,
                  O_AlarmABCondition => #OverCurrentHAlmCond,
                  O_HHHReached => "NotUsedBool",
                  O_HHReached => "NotUsedBool",
                  O_HReached => "NotUsedBool",
                  O_LReached => "NotUsedBool",
                  O_LLReached => "NotUsedBool",
                  O_LLLReached => "NotUsedBool",
                  H_IAnim => #"H_GBChain2W1S-FC302PN".H_MotorCurrentIAnim[1].H_DWord);
END_REGION

REGION Network 23: **** 7.1 - Submodule - Non-Machine **** Transfer IN Set
   // Transfer IN Set
   IF "TRUE" THEN
       #_LTrfInSet(I_AnyDet := #I_EntranceDet,   // "LGBTrfIn"
                   I_StopDet := #I_EntranceDet AND NOT #I_StopDetPrev,
                   I_LocalPB := #I_PBSet,
                   I_ManInfeedAllowed := #I_ManInfeedAllowedSet,
                   I_TrfInBegin := #I_TrfInSetBegin,
                   I_InterlockOk := #I_TrfInSetIntlkOk,
                   I_ReadyForOperation := #FrqReadyForOperationMot,
                   I_TrfInRdyDlv := #I_TrfInSetRdyDlv,
                   I_TrfInOutfeedHold := "FALSE",
                   I_TrfInTM := #I_TrfInSetTM,
                   I_TrfOutTM := "FALSE",
                   I_ProductionStop := #IO_Modes.LProductionMode.ProdStpMode OR #IO_Modes.LProductionMode.ProdStpModeSel,
                   I_TrainCond := #C_Config.TrainActivatedSet,
                   I_EnableAlarm := #C_Config.EnableAlarmTransfer,
                   I_ForcedMan := #IO_Modes.LMode.ForcedMan,
                   I_GenRevSw := #IO_Modes.LGeneralFunc.GenRevSwitch,
                   I_GeneralPB := #IO_Modes.LMode.SetPBMan,
                   IO_Modes := #IO_Modes,
                   H_HMI := #H_HMITrfInSet,
                   H_TrfIn := #"H_GBChain2W1S-FC302PN".H_TrfInSet,
                   H_FncSelInHMI := #H_FncSelInHMI,
                   C_TrfInUsed := #C_Config.TrfInSetUsed,
                   O_TrfInCmd => #TrfInSetCmd,
                   O_TrfInRdyRcv => #TrfInSetRdyRcv,
                   O_TrfInInfeedHold => #TrfInfeedHoldSet,
                   O_TrfInArrived => #TrfInSetArrived,
                   O_StopTrfOutCmd => #StopTrfOutSetCmd,
                   O_TrfInActive => #TrfInSetActive,
                   O_TrfInFinished => #TrfInSetFinished,
                   O_InterlockAlarm => #AD_TrfInSetInterlock);
   END_IF;
END_REGION

REGION Network 24: **** 7.1 - Submodule - Non-Machine **** Transfer Out Set
   // Transfer Out Set
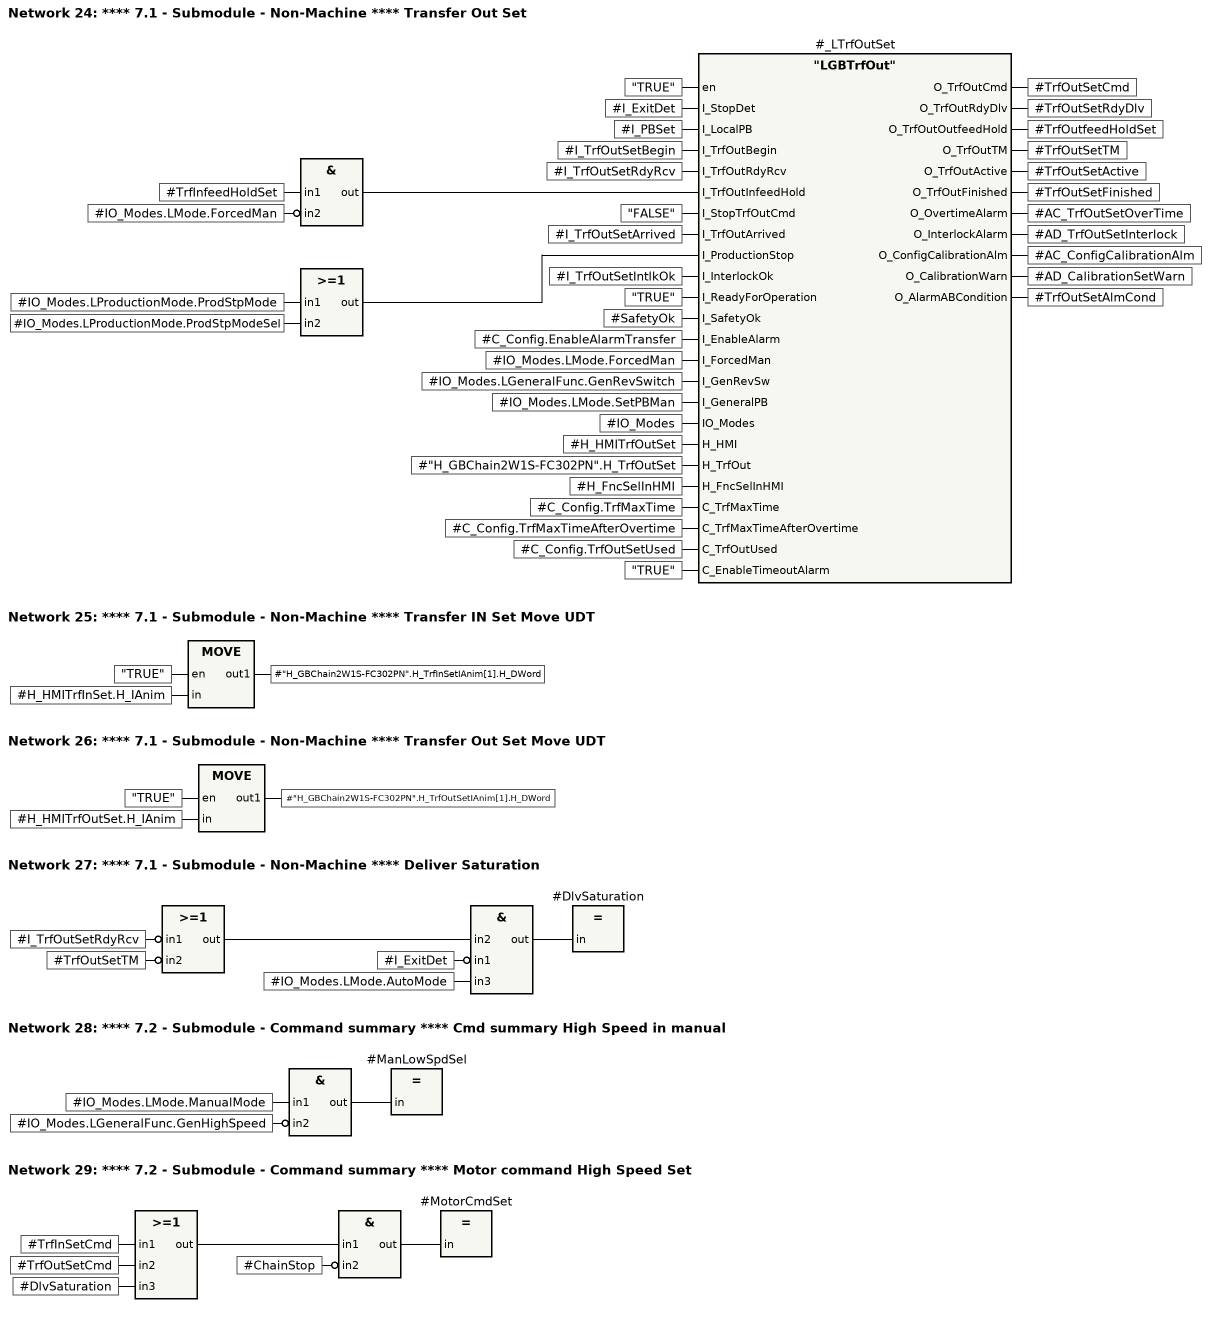
   IF "TRUE" THEN
       #_LTrfOutSet(I_StopDet := #I_ExitDet,   // "LGBTrfOut"
                    I_LocalPB := #I_PBSet,
                    I_TrfOutBegin := #I_TrfOutSetBegin,
                    I_TrfOutRdyRcv := #I_TrfOutSetRdyRcv,
                    I_TrfOutInfeedHold := #TrfInfeedHoldSet AND NOT #IO_Modes.LMode.ForcedMan,
                    I_StopTrfOutCmd := "FALSE",
                    I_TrfOutArrived := #I_TrfOutSetArrived,
                    I_ProductionStop := #IO_Modes.LProductionMode.ProdStpMode OR #IO_Modes.LProductionMode.ProdStpModeSel,
                    I_InterlockOk := #I_TrfOutSetIntlkOk,
                    I_ReadyForOperation := "TRUE",
                    I_SafetyOk := #SafetyOk,
                    I_EnableAlarm := #C_Config.EnableAlarmTransfer,
                    I_ForcedMan := #IO_Modes.LMode.ForcedMan,
                    I_GenRevSw := #IO_Modes.LGeneralFunc.GenRevSwitch,
                    I_GeneralPB := #IO_Modes.LMode.SetPBMan,
                    IO_Modes := #IO_Modes,
                    H_HMI := #H_HMITrfOutSet,
                    H_TrfOut := #"H_GBChain2W1S-FC302PN".H_TrfOutSet,
                    H_FncSelInHMI := #H_FncSelInHMI,
                    C_TrfMaxTime := #C_Config.TrfMaxTime,
                    C_TrfMaxTimeAfterOvertime := #C_Config.TrfMaxTimeAfterOvertime,
                    C_TrfOutUsed := #C_Config.TrfOutSetUsed,
                    C_EnableTimeoutAlarm := "TRUE",
                    O_TrfOutCmd => #TrfOutSetCmd,
                    O_TrfOutRdyDlv => #TrfOutSetRdyDlv,
                    O_TrfOutOutfeedHold => #TrfOutfeedHoldSet,
                    O_TrfOutTM => #TrfOutSetTM,
                    O_TrfOutActive => #TrfOutSetActive,
                    O_TrfOutFinished => #TrfOutSetFinished,
                    O_OvertimeAlarm => #AC_TrfOutSetOverTime,
                    O_InterlockAlarm => #AD_TrfOutSetInterlock,
                    O_ConfigCalibrationAlm => #AC_ConfigCalibrationAlm,
                    O_CalibrationWarn => #AD_CalibrationSetWarn,
                    O_AlarmABCondition => #TrfOutSetAlmCond);
   END_IF;
END_REGION

REGION Network 25: **** 7.1 - Submodule - Non-Machine **** Transfer IN Set Move UDT
   // Transfer IN Set Move UDT
   IF "TRUE" THEN #"H_GBChain2W1S-FC302PN".H_TrfInSetIAnim[1].H_DWord := #H_HMITrfInSet.H_IAnim; END_IF;
END_REGION

REGION Network 26: **** 7.1 - Submodule - Non-Machine **** Transfer Out Set Move UDT
   // Transfer Out Set Move UDT
   IF "TRUE" THEN #"H_GBChain2W1S-FC302PN".H_TrfOutSetIAnim[1].H_DWord := #H_HMITrfOutSet.H_IAnim; END_IF;
END_REGION

REGION Network 27: **** 7.1 - Submodule - Non-Machine **** Deliver Saturation
   #DlvSaturation := (NOT #I_TrfOutSetRdyRcv OR NOT #TrfOutSetTM) AND NOT #I_ExitDet AND #IO_Modes.LMode.AutoMode;
END_REGION

REGION Network 28: **** 7.2 - Submodule - Command summary **** Cmd summary High Speed in manual
   // Cmd summary High Speed in manual
   #ManLowSpdSel := #IO_Modes.LMode.ManualMode AND NOT #IO_Modes.LGeneralFunc.GenHighSpeed;
END_REGION

REGION Network 29: **** 7.2 - Submodule - Command summary **** Motor command High Speed Set
   // Motor command High Speed Set
   #MotorCmdSet := (#TrfInSetCmd OR #TrfOutSetCmd OR #DlvSaturation) AND NOT #ChainStop;
END_REGION

REGION Network 30: **** 7.2 - Submodule - Command summary **** Motor command Reset
   // Motor command Reset
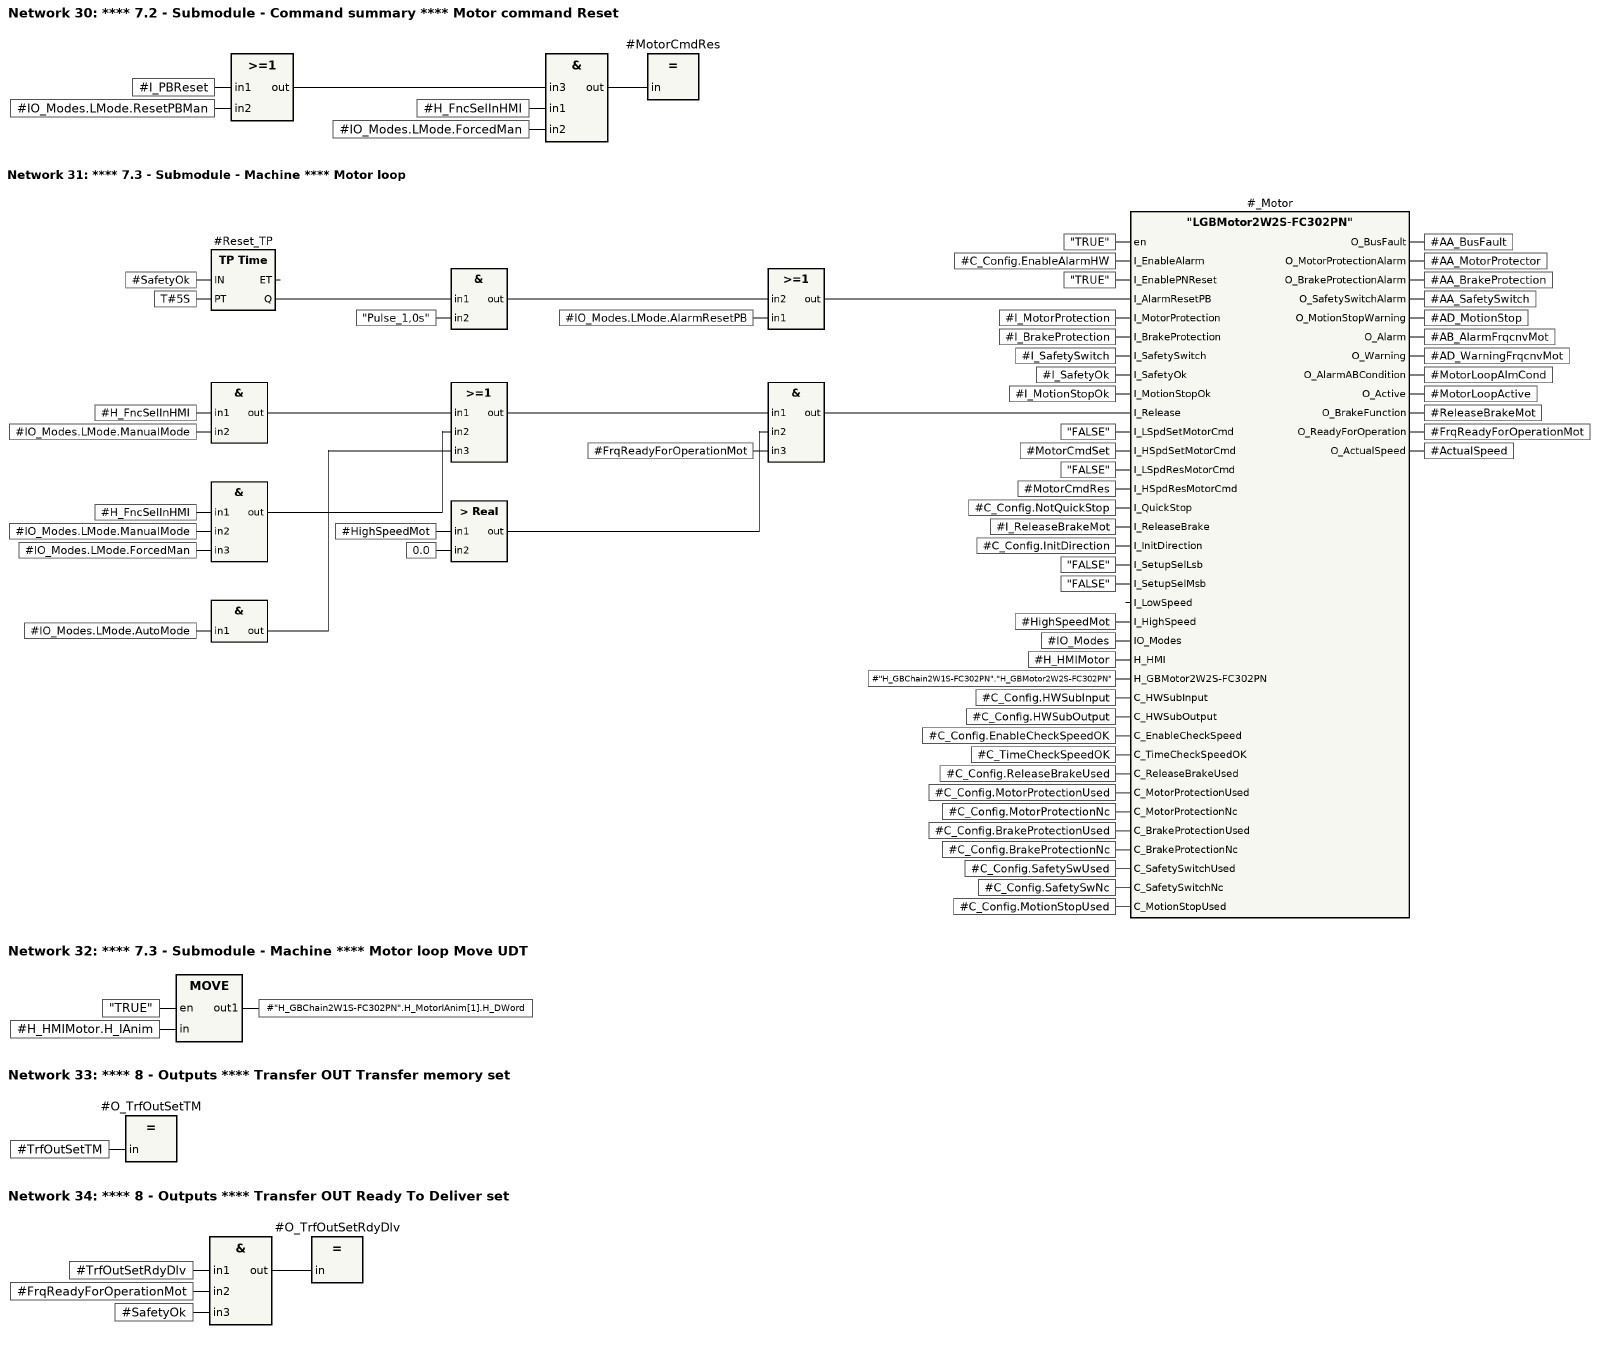
   #MotorCmdRes := (#I_PBReset OR #IO_Modes.LMode.ResetPBMan) AND #H_FncSelInHMI AND #IO_Modes.LMode.ForcedMan;
END_REGION

REGION Network 31: **** 7.3 - Submodule - Machine **** Motor loop
   #Reset_TP(IN := #SafetyOk, PT := T#5S);   // TP
   IF "TRUE" THEN
       #_Motor(I_EnableAlarm := #C_Config.EnableAlarmHW,   // "LGBMotor2W2S-FC302PN"
               I_EnablePNReset := "TRUE",
               I_AlarmResetPB := (#Reset_TP.Q AND "Pulse_1,0s") OR #IO_Modes.LMode.AlarmResetPB,
               I_MotorProtection := #I_MotorProtection,
               I_BrakeProtection := #I_BrakeProtection,
               I_SafetySwitch := #I_SafetySwitch,
               I_SafetyOk := #I_SafetyOk,
               I_MotionStopOk := #I_MotionStopOk,
               I_Release := ((#H_FncSelInHMI AND #IO_Modes.LMode.ManualMode) OR (#H_FncSelInHMI AND #IO_Modes.LMode.ManualMode AND #IO_Modes.LMode.ForcedMan) OR #IO_Modes.LMode.AutoMode) AND (#HighSpeedMot > 0.0) AND #FrqReadyForOperationMot,
               I_LSpdSetMotorCmd := "FALSE",
               I_HSpdSetMotorCmd := #MotorCmdSet,
               I_LSpdResMotorCmd := "FALSE",
               I_HSpdResMotorCmd := #MotorCmdRes,
               I_QuickStop := #C_Config.NotQuickStop,
               I_ReleaseBrake := #I_ReleaseBrakeMot,
               I_InitDirection := #C_Config.InitDirection,
               I_SetupSelLsb := "FALSE",
               I_SetupSelMsb := "FALSE",
               I_HighSpeed := #HighSpeedMot,
               IO_Modes := #IO_Modes,
               H_HMI := #H_HMIMotor,
               "H_GBMotor2W2S-FC302PN" := #"H_GBChain2W1S-FC302PN"."H_GBMotor2W2S-FC302PN",
               C_HWSubInput := #C_Config.HWSubInput,
               C_HWSubOutput := #C_Config.HWSubOutput,
               C_EnableCheckSpeed := #C_Config.EnableCheckSpeedOK,
               C_TimeCheckSpeedOK := #C_TimeCheckSpeedOK,
               C_ReleaseBrakeUsed := #C_Config.ReleaseBrakeUsed,
               C_MotorProtectionUsed := #C_Config.MotorProtectionUsed,
               C_MotorProtectionNc := #C_Config.MotorProtectionNc,
               C_BrakeProtectionUsed := #C_Config.BrakeProtectionUsed,
               C_BrakeProtectionNc := #C_Config.BrakeProtectionNc,
               C_SafetySwitchUsed := #C_Config.SafetySwUsed,
               C_SafetySwitchNc := #C_Config.SafetySwNc,
               C_MotionStopUsed := #C_Config.MotionStopUsed,
               O_BusFault => #AA_BusFault,
               O_MotorProtectionAlarm => #AA_MotorProtector,
               O_BrakeProtectionAlarm => #AA_BrakeProtection,
               O_SafetySwitchAlarm => #AA_SafetySwitch,
               O_MotionStopWarning => #AD_MotionStop,
               O_Alarm => #AB_AlarmFrqcnvMot,
               O_Warning => #AD_WarningFrqcnvMot,
               O_AlarmABCondition => #MotorLoopAlmCond,
               O_Active => #MotorLoopActive,
               O_BrakeFunction => #ReleaseBrakeMot,
               O_ReadyForOperation => #FrqReadyForOperationMot,
               O_ActualSpeed => #ActualSpeed);
   END_IF;
END_REGION

REGION Network 32: **** 7.3 - Submodule - Machine **** Motor loop Move UDT
   IF "TRUE" THEN #"H_GBChain2W1S-FC302PN".H_MotorIAnim[1].H_DWord := #H_HMIMotor.H_IAnim; END_IF;
END_REGION

REGION Network 33: **** 8 - Outputs **** Transfer OUT Transfer memory set
   // Transfer OUT Transfer memory set
   #O_TrfOutSetTM := #TrfOutSetTM;
END_REGION

REGION Network 34: **** 8 - Outputs **** Transfer OUT Ready To Deliver set
   // Transfer OUT Ready To Deliver set
   #O_TrfOutSetRdyDlv := #TrfOutSetRdyDlv AND #FrqReadyForOperationMot AND #SafetyOk;
END_REGION

REGION Network 35: **** 8 - Outputs **** Transfer IN Arrived set
   // Transfer IN Arrived set
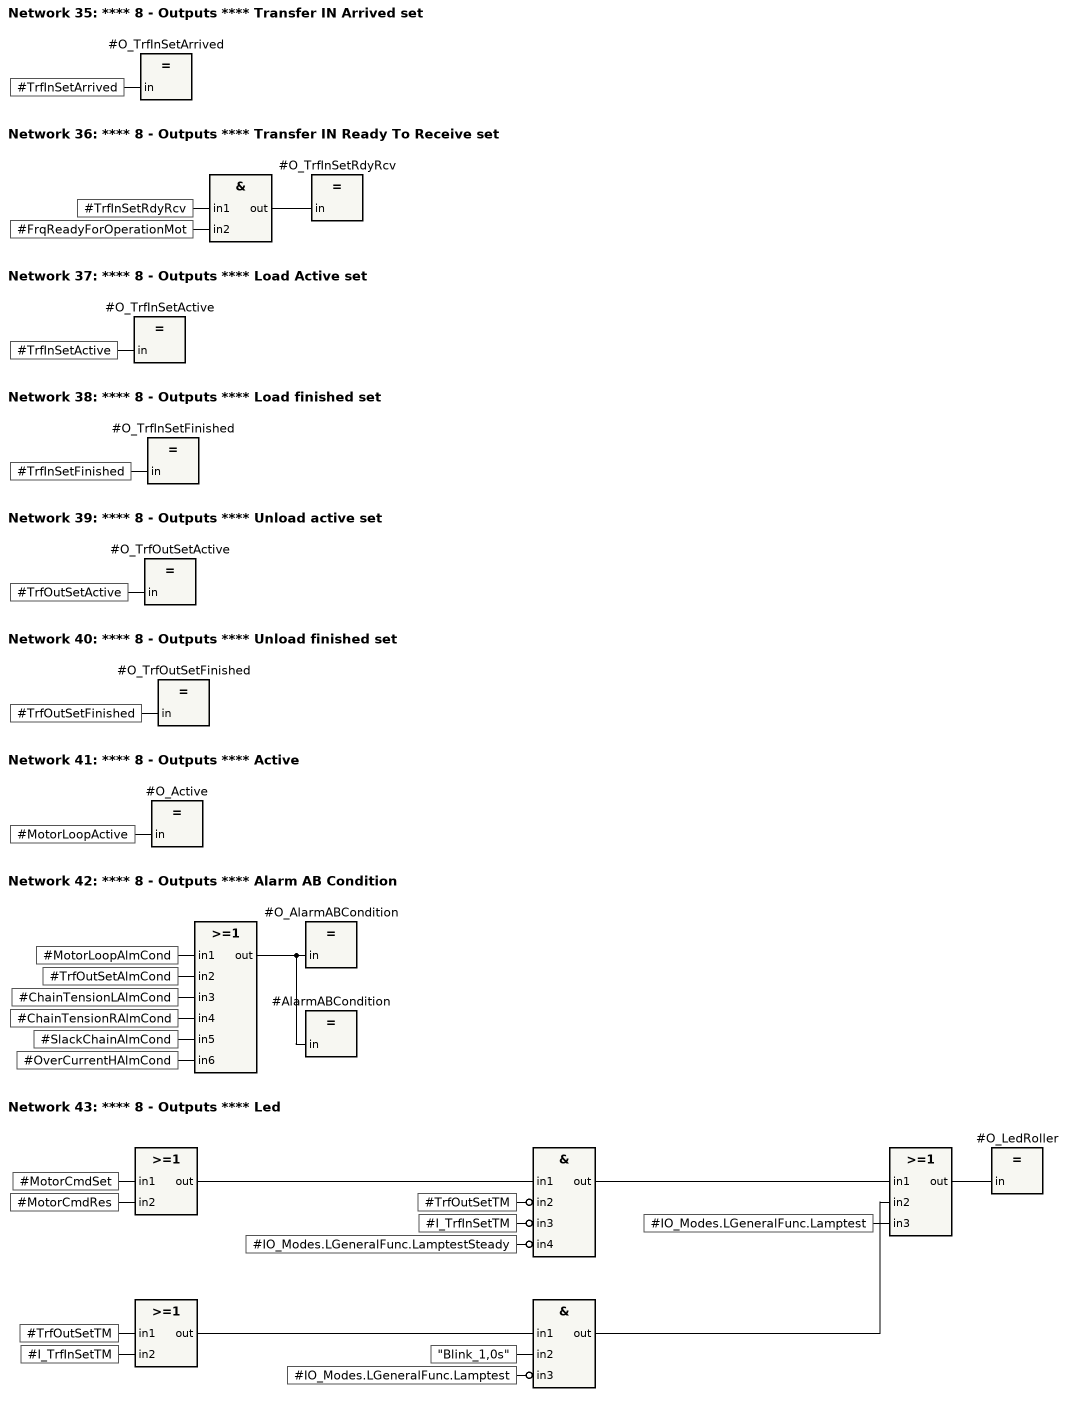
   #O_TrfInSetArrived := #TrfInSetArrived;
END_REGION

REGION Network 36: **** 8 - Outputs **** Transfer IN Ready To Receive set
   // Transfer IN Ready To Receive set
   #O_TrfInSetRdyRcv := #TrfInSetRdyRcv AND #FrqReadyForOperationMot;
END_REGION

REGION Network 37: **** 8 - Outputs **** Load Active set
   // Load Active set
   #O_TrfInSetActive := #TrfInSetActive;
END_REGION

REGION Network 38: **** 8 - Outputs **** Load finished set
   // Load finished set
   #O_TrfInSetFinished := #TrfInSetFinished;
END_REGION

REGION Network 39: **** 8 - Outputs **** Unload active set
   // Unload active set
   #O_TrfOutSetActive := #TrfOutSetActive;
END_REGION

REGION Network 40: **** 8 - Outputs **** Unload finished set
   // Unload finished set
   #O_TrfOutSetFinished := #TrfOutSetFinished;
END_REGION

REGION Network 41: **** 8 - Outputs **** Active
   // Active
   #O_Active := #MotorLoopActive;
END_REGION

REGION Network 42: **** 8 - Outputs **** Alarm AB Condition
   // Alarm AB Condition
   #O_AlarmABCondition := #MotorLoopAlmCond OR #TrfOutSetAlmCond OR #ChainTensionLAlmCond OR #ChainTensionRAlmCond OR #SlackChainAlmCond OR #OverCurrentHAlmCond;
   #AlarmABCondition := #O_AlarmABCondition;
END_REGION

REGION Network 43: **** 8 - Outputs **** Led
   // Led
   #O_LedRoller := ((#MotorCmdSet OR #MotorCmdRes) AND NOT #TrfOutSetTM AND NOT #I_TrfInSetTM AND NOT #IO_Modes.LGeneralFunc.LamptestSteady) OR ((#TrfOutSetTM OR #I_TrfInSetTM) AND "Blink_1,0s" AND NOT #IO_Modes.LGeneralFunc.Lamptest) OR #IO_Modes.LGeneralFunc.Lamptest;
END_REGION

REGION Network 44: **** 8 - Outputs **** Occupied
   // Occupied
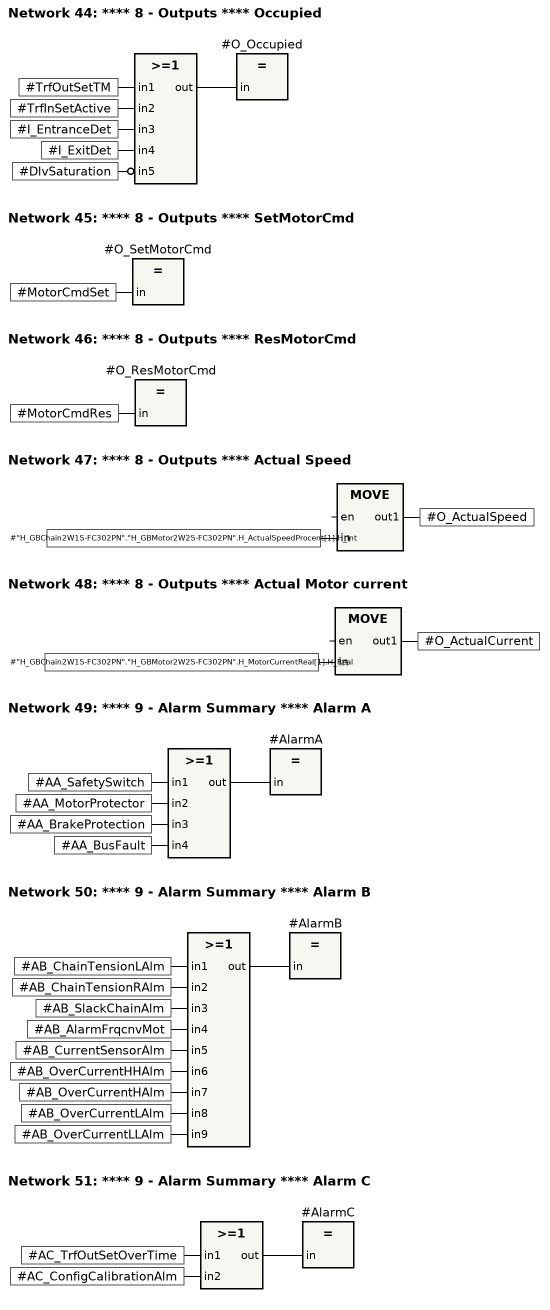
   #O_Occupied := #TrfOutSetTM OR #TrfInSetActive OR #I_EntranceDet OR #I_ExitDet OR NOT #DlvSaturation;
END_REGION

REGION Network 45: **** 8 - Outputs **** SetMotorCmd
   // SetMotorCmd
   #O_SetMotorCmd := #MotorCmdSet;
END_REGION

REGION Network 46: **** 8 - Outputs **** ResMotorCmd
   // ResMotorCmd
   #O_ResMotorCmd := #MotorCmdRes;
END_REGION

REGION Network 47: **** 8 - Outputs **** Actual Speed
   #O_ActualSpeed := #"H_GBChain2W1S-FC302PN"."H_GBMotor2W2S-FC302PN".H_ActualSpeedProcent[1].H_Int;
END_REGION

REGION Network 48: **** 8 - Outputs **** Actual Motor current
   #O_ActualCurrent := #"H_GBChain2W1S-FC302PN"."H_GBMotor2W2S-FC302PN".H_MotorCurrentReal[1].H_Real;
END_REGION

REGION Network 49: **** 9 - Alarm Summary **** Alarm A
   // Alarm A
   #AlarmA := #AA_SafetySwitch OR #AA_MotorProtector OR #AA_BrakeProtection OR #AA_BusFault;
END_REGION

REGION Network 50: **** 9 - Alarm Summary **** Alarm B
   // Alarm B
   #AlarmB := #AB_ChainTensionLAlm OR #AB_ChainTensionRAlm OR #AB_SlackChainAlm OR #AB_AlarmFrqcnvMot OR #AB_CurrentSensorAlm OR #AB_OverCurrentHHAlm OR #AB_OverCurrentHAlm OR #AB_OverCurrentLAlm OR #AB_OverCurrentLLAlm;
END_REGION

REGION Network 51: **** 9 - Alarm Summary **** Alarm C
   // Alarm C
   #AlarmC := #AC_TrfOutSetOverTime OR #AC_ConfigCalibrationAlm;
END_REGION

REGION Network 52: **** 9 - Alarm Summary **** Alarm D
   // Alarm D
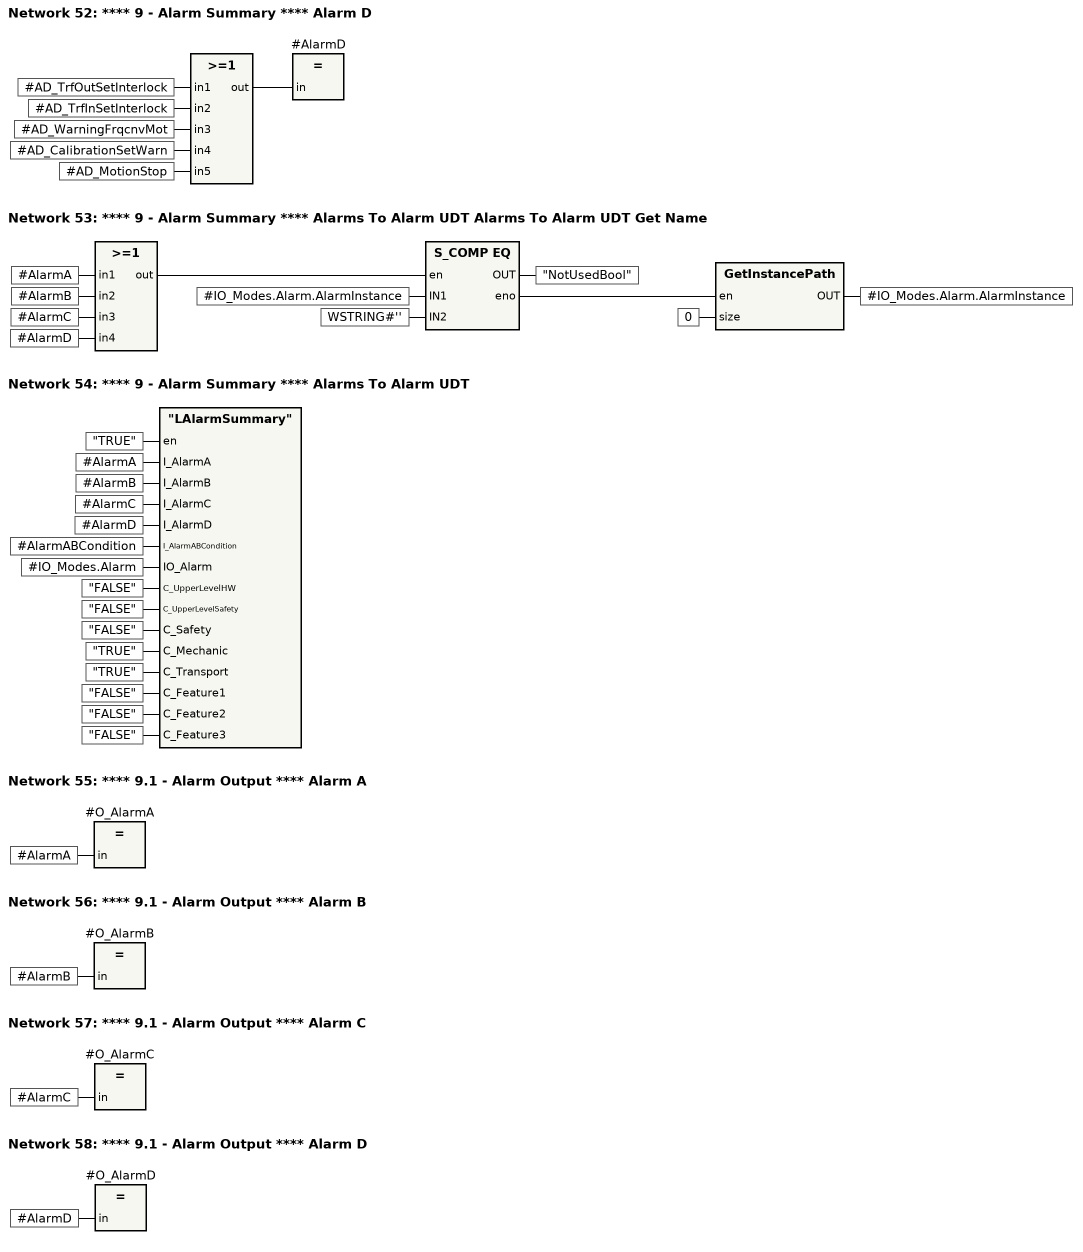
   #AlarmD := #AD_TrfOutSetInterlock OR #AD_TrfInSetInterlock OR #AD_WarningFrqcnvMot OR #AD_CalibrationSetWarn OR #AD_MotionStop;
END_REGION

REGION Network 53: **** 9 - Alarm Summary **** Alarms To Alarm UDT Alarms To Alarm UDT Get Name
   // Alarm D
   S_COMP(EN := #AlarmA OR #AlarmB OR #AlarmC OR #AlarmD,
          IN1 := #IO_Modes.Alarm.AlarmInstance,
          IN2 := WSTRING#'',
          OUT => "NotUsedBool",
          ENO => #_w1);
   IF #_w1 THEN GetInstancePath(size := 0, OUT => #IO_Modes.Alarm.AlarmInstance); END_IF;
END_REGION

REGION Network 54: **** 9 - Alarm Summary **** Alarms To Alarm UDT
   // Alarm D
   IF "TRUE" THEN
       "LAlarmSummary"(I_AlarmA := #AlarmA,
                       I_AlarmB := #AlarmB,
                       I_AlarmC := #AlarmC,
                       I_AlarmD := #AlarmD,
                       I_AlarmABCondition := #AlarmABCondition,
                       IO_Alarm := #IO_Modes.Alarm,
                       C_UpperLevelHW := "FALSE",
                       C_UpperLevelSafety := "FALSE",
                       C_Safety := "FALSE",
                       C_Mechanic := "TRUE",
                       C_Transport := "TRUE",
                       C_Feature1 := "FALSE",
                       C_Feature2 := "FALSE",
                       C_Feature3 := "FALSE");
   END_IF;
END_REGION

REGION Network 55: **** 9.1 - Alarm Output **** Alarm A
   // Alarm A
   #O_AlarmA := #AlarmA;
END_REGION

REGION Network 56: **** 9.1 - Alarm Output **** Alarm B
   // Alarm B
   #O_AlarmB := #AlarmB;
END_REGION

REGION Network 57: **** 9.1 - Alarm Output **** Alarm C
   // Alarm C
   #O_AlarmC := #AlarmC;
END_REGION

REGION Network 58: **** 9.1 - Alarm Output **** Alarm D
   // Alarm D
   #O_AlarmD := #AlarmD;
END_REGION

REGION Network 59: **** 9.2 - Alarm DWord**** Alarm To DWord
   // Alarm Word
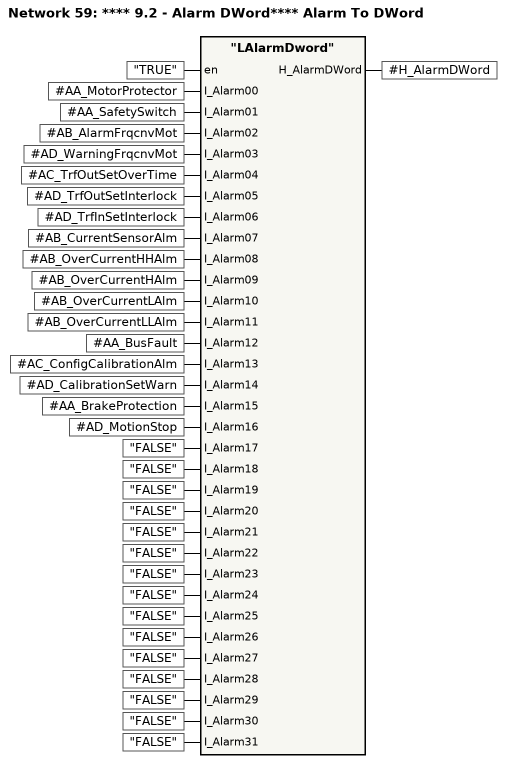
   IF "TRUE" THEN
       "LAlarmDword"(I_Alarm00 := #AA_MotorProtector,
                     I_Alarm01 := #AA_SafetySwitch,
                     I_Alarm02 := #AB_AlarmFrqcnvMot,
                     I_Alarm03 := #AD_WarningFrqcnvMot,
                     I_Alarm04 := #AC_TrfOutSetOverTime,
                     I_Alarm05 := #AD_TrfOutSetInterlock,
                     I_Alarm06 := #AD_TrfInSetInterlock,
                     I_Alarm07 := #AB_CurrentSensorAlm,
                     I_Alarm08 := #AB_OverCurrentHHAlm,
                     I_Alarm09 := #AB_OverCurrentHAlm,
                     I_Alarm10 := #AB_OverCurrentLAlm,
                     I_Alarm11 := #AB_OverCurrentLLAlm,
                     I_Alarm12 := #AA_BusFault,
                     I_Alarm13 := #AC_ConfigCalibrationAlm,
                     I_Alarm14 := #AD_CalibrationSetWarn,
                     I_Alarm15 := #AA_BrakeProtection,
                     I_Alarm16 := #AD_MotionStop,
                     I_Alarm17 := "FALSE",
                     I_Alarm18 := "FALSE",
                     I_Alarm19 := "FALSE",
                     I_Alarm20 := "FALSE",
                     I_Alarm21 := "FALSE",
                     I_Alarm22 := "FALSE",
                     I_Alarm23 := "FALSE",
                     I_Alarm24 := "FALSE",
                     I_Alarm25 := "FALSE",
                     I_Alarm26 := "FALSE",
                     I_Alarm27 := "FALSE",
                     I_Alarm28 := "FALSE",
                     I_Alarm29 := "FALSE",
                     I_Alarm30 := "FALSE",
                     I_Alarm31 := "FALSE",
                     H_AlarmDWord => #H_AlarmDWord);
   END_IF;
END_REGION
END_FUNCTION_BLOCK
